TYPE TYP_VESSEL_HW :
STRUCT
	In : TYP_VESSEL_HW_IN;
	Out : TYP_VESSEL_HW_OUT;
END_STRUCT
END_TYPE

(* stored: Version 1.1.0.1, ProductVersion 3.1.4024.12
   DUT TYP_VESSEL_HW: Id {3d38f663-91d0-4442-9cb9-0881129e3f7c} *)
